// TwinCAT 3 PLC project Warehouse_Extended
// ProgramVersion: 3.1.4026.16
// libraries:
//   Tc2_Standard, * (Beckhoff Automation GmbH)
//   Tc2_System, * (Beckhoff Automation GmbH)
// project tree:
//   / GlobalTextList.TcGTLO, PlcTask.TcTTO
//   POUs/ FB_WarehouseStock.TcPOU, MAIN.TcPOU
// real-time tasks:
//   TASK PlcTask: cycle T#10ms, priority 20, ADS port 351

CONFIGURATION Warehouse_Extended
    RESOURCE PLC ON TwinCAT3
        TASK PlcTask(INTERVAL := T#10ms, PRIORITY := 20);
        PROGRAM MAIN WITH PlcTask : MAIN;
    END_RESOURCE
END_CONFIGURATION

// ---- POUs/MAIN.TcPOU
PROGRAM MAIN
VAR
	iProductNumber:			INT;			//Eingabe der ein- oder auszulagernder Produktenummer
	bStartStore: 			BOOL;			//Taster um Einlagerung zu starten
	bStartRemove:			BOOL;			//Taster um Auslagerung zu starten
	bLastCLKStartStore:		BOOL;			//Zwischenspeicher des letzten Zustandes von StartStore für Flankenerkennung
	bLastCLKStartRemove: 	BOOL;			//Zwischenspeicher des letzten Zustandes von StartRemove für Flankenerkennung
	Warehouse:				FB_WarehouseStock;
END_VAR

{region "store"}
IF bStartStore AND NOT bLastCLKStartStore THEN
	Warehouse.M_Store(iProdNumber := iProductNumber);
END_IF
{endregion}

{region "remove"}
IF bStartRemove AND NOT bLastCLKStartRemove THEN
	Warehouse.M_Remove(iProdNumber := iProductNumber);
END_IF
{endregion}

bLastCLKStartStore 		:= bStartStore;
bLastCLKStartRemove 	:= bStartRemove;

END_PROGRAM

// ---- POUs/FB_WarehouseStock.TcPOU
FUNCTION_BLOCK FB_WarehouseStock
VAR_INPUT	
END_VAR
VAR_OUTPUT
END_VAR
VAR
	iXAxis:			INT;
	iYAxis:			INT;
	bStored:			BOOL;
	bRemoved:			BOOL;
	arrStockPosition:	ARRAY[1..7, 1..12] OF INT;
END_VAR

METHOD M_Remove : BOOL
VAR_INPUT
	iProdNumber: 		INT;
END_VAR
bRemoved := FALSE;

IF iProdNumber = 0 THEN
	RETURN;
END_IF

FOR iXAxis := 1 TO 7 BY 1 DO
	FOR iYAxis :=  1 TO 12 BY 1 DO
		IF arrStockPosition[iXAxis, iYAxis] = iProdNumber THEN
			arrStockPosition[iXAxis, iYAxis] := 0;
			bRemoved := TRUE;
			EXIT;
		END_IF
		IF bRemoved = TRUE THEN
			RETURN;
		END_IF
	END_FOR
END_FOR
END_METHOD

METHOD M_Store : BOOL
VAR_INPUT
	iProdNumber: 		INT;
END_VAR
bStored := FALSE;

IF iProdNumber = 0 THEN
	RETURN;
END_IF

FOR iXAxis := 1 TO 7 BY 1 DO
	FOR iYAxis :=  1 TO 12 BY 1 DO
		IF arrStockPosition[iXAxis, iYAxis] = 0 THEN
			arrStockPosition[iXAxis, iYAxis] := iProdNumber;
			bStored := TRUE;
			EXIT;
		END_IF
		IF bStored = TRUE THEN
			RETURN;
		END_IF
	END_FOR
END_FOR
END_METHOD

END_FUNCTION_BLOCK
